(*

.. <legal notes>

legal notes
=================
| SPDX-FileCopyrightText: © 2026 Oleksandr Tiutyk <trofimich@gmail.com>
| SPDX-License-Identifier: LGPL-3.0-only
| For details check: LGPL-3.0-only_

.. _LGPL-3.0-only: https://www.gnu.org/licenses/lgpl-3.0.en.html

.. </legal notes>

*)

FUNCTION_BLOCK INTERNAL NamespaceExtractor
VAR_OUTPUT
	{attribute 'init_namespace'} 
	CurrentNamespace : STRING(255);	
END_VAR

END_FUNCTION_BLOCK

(* stored: Version 1.1.0.1
   POU NamespaceExtractor: Id {ec6d51c5-289a-48c0-9421-d9f46a88f34e}, SpecialFunc None *)
